INTERFACE I_WordBuilder EXTENDS T_QueryInterface

END_INTERFACE

(* stored: Version 1.1.0.1, ProductVersion 3.1.4024.4
   Itf I_WordBuilder: Id {7b4ee324-8ed2-4db6-b403-fd2982d425cd} *)
